TYPE E_HostCmdId :
(
    None        := 0,
    StartAuto   := 1,
    Pause       := 2,
    ContinueRun := 3,
    Stop        := 4,
    Reset       := 5,
    ClearAlarm  := 6,
    HomeAll     := 7,
    ToManual    := 8,
    ToAuto      := 9,
    ManualAct   := 10
);
END_TYPE

(* stored: Version 1.1.0.1, ProductVersion 3.1.4026.18
   DUT E_HostCmdId: Id {ab1ca3fa-4211-491b-a67a-2f9fae77ffac} *)
